{attribute 'GeneratedUsingTerminal: KL2631'}
{attribute addProperty BoxType "KL2631"}
{attribute addProperty Id "Channel_1AT %Q*Channel_460B8C400"}
{attribute addProperty CRC "3732460390"}
{attribute addProperty Size "0"}
TYPE KL2631_DE78D366 :
STRUCT
	{attribute addProperty Name "Channel_1"}
	Channel_1 : Channel_460B8C40;
END_STRUCT
END_TYPE

(* stored: Version 1.2.0.0, ProductVersion 3.1.4024.9
   DUT KL2631_DE78D366: Id {7dbbf79f-347c-45b2-913b-e53fa3213fbd} *)
